// TIA Portal V18 export
// export: Created 2026-01-09T11:23:42.865511Z, ExportSetting WithDefaults, DisplayName Totally Integrated Automation Portal, DisplayVersion V18 Update 5, DisplayName TIA Portal Openness, DisplayVersion V18 Update 5, DisplayName TIA Portal Teamcenter Gateway, DisplayVersion V18, DisplayName TIA Portal Version Control Interface, DisplayVersion V18, DisplayName SINAMICS Startdrive Advanced, DisplayVersion V18 SP2 Update 1, DisplayName SINAMICS Startdrive G110M, G120, G120C, G120D, G120P, G115D, DisplayVersion V18 SP2 Update 1, DisplayName SINAMICS Startdrive G130, G150, S120, S150, SINAMICS MV, S210, G220, S200, DisplayVersion V18 SP2 Update 1, DisplayName STEP 7 Professional, DisplayVersion V18 Update 5, DisplayName STEP 7 Safety, DisplayVersion V18, DisplayName WinCC Professional, DisplayVersion V18 Update 5
Screen "820 User"  1280x800, Number=820, Template=08CtrlPanel
  ScreenLayer "Layer_0"
    UserView "用户视图_1" at 0,85 size 1278x605  Appearance=Appearance3D, CountVisibleItems=8, ViewType=ViewTypeComplex, StyleItem=Benutzeranzeige
    Button "btnMenu5_1" at 384,725 size 128x75  Mode=Text, Authorization=User administration, StyleItem=BtnActive20, TextOff="用户设定 / User Config / Užívateľ Konfigurácia"
      on Click: ActivateScreen(Screen name := , Object number := 0); SetTag(Tag := Sys_VersionManagement_HMIPageID, Value := 820)
